TEXTLIST PositionType
  0 = 'Absolute'
  1 = 'Relative'
   = ''
END_TEXTLIST

(* stored: Version 1.1.0.1
   TextList PositionType: Id {30202f4d-baa7-4704-bc25-6086c5d218c3} *)
